FUNCTION_BLOCK SLIDER (* recognize bubble size *)
  (* Version 1.0, AN, SWDC RTSoft *)
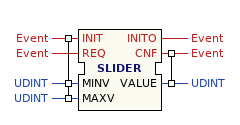
  EVENT_INPUT
    INIT WITH MINV, MAXV;
  END_EVENT
  EVENT_OUTPUT
    INITO;
    CNF WITH VALUE;
  END_EVENT
  VAR_INPUT
    MINV : UDINT;
    MAXV : UDINT;
  END_VAR
  VAR_OUTPUT
    VALUE : UDINT;
  END_VAR
END_FUNCTION_BLOCK
(* other elements stored in the file *)
(* Event Name=REQ Type=Event *)
